// TIA Portal V19 export
FUNCTION "TetraPakV50_9" : Void   // FC118, STL
TITLE = Tetra Pak V50 IO-Link DeviceID 9 Process Data
{ S7_Optimized_Access := 'TRUE' }
AUTHOR : AFL
FAMILY : IO_Link
NAME : TP_V50_9
// Data words uses in function
// 
// HMI_CMD, dw X - command word from SCADA
// Bit 0 = auto
// Bit 1 = Manuel deactivate
// Bit 2 = Manuel activate
// Bit 3 = Locate
// Bit 4 = spare
// Bit 5 = spare
// Bit 6 = spare
// 
// HMI_INFO, dw X - info word to SCADA
// Bit 0  = activated
// Bit 1  = changing
// Bit 2  = faulty 
// Bit 3  = auto_man, Manuel = 1 
// Bit 4  = man_on_off
// Bit 5  = Reset_FB
// Bit 6  = ManualSelected
// Bit 7  = Set_FB
// Bit 8  = Locate Active 
// Bit 9  = spare 
// Bit 10 = spare 
// Bit 11 = spare  
// Bit 12 = spare 
// Bit 13 = spare 
// Bit 14 = fb_error - Alarm feedback error
// Bit 15 = spare 
// 
// Error status
// 0 (Everything is OK)
// 16 (Sensor target missing (#16))
// 17 (Setup prerequisite issue (#17))
// 18 (Pneumatic part issue (#18))
// 19 (Seat lift sensor issue (#19))
// 20 (Position not reached (#20))
// 21 (Unexpected movement (#21))
// 22 (Seat-lift sensor missing (#22))
// 23 (Pilot valve 1 missing (#23))
// 24 (Pilot valve 2 missing (#24))
// 25 (Pilot valve 3 missing (#25))
// 26 (Interlock active (#26))
// 27 (Output short circuit (#27))
// 28 (Setup aborted (#28))
// 29 (Blocked button (#29))
// 30 (Communication failure (#30))
// 31 (Safety stop active (#31))
// stored: AutoNumber false
   VAR_INPUT
      Addr : Int;   // First Byte address of 4 byte address space
      Pulse : Bool;   // Trigger one clean pulse on SV 1
      SV_1 : Bool;   // Trigger solenoid valve 1 for main valve activation
      Wink : Bool;   // Visual indication for locating the unit
   END_VAR
   VAR_OUTPUT
      ValvePosition : Real;   // Current Valve position (0 to 720 * 0.1)
      ValveState : Bool;   // Current Valve state
      O_DI4 : Bool;   // Output signal status Pin 4
      O_DI2 : Bool;   // Output signal status Pin 2
      Teach : Bool;   // Teach output for teach command bit
   END_VAR
   VAR_IN_OUT
      itemInfo : "ItemInfo_UDT";
      itemCommand : "ItemCommand_UDT";
      ErrorStatus : Byte;   // See Block Comment
      Main : Bool;   // Main energised Position
      DE_EN : Bool;   // De-Energized
      O_DA : Bool;   // Output device recognised
      O_DE : Bool;   // Output device error event has appeared
      O_PQ : Bool;   // Output port qualifer proces data valid
   END_VAR
   VAR_TEMP
      TW_Flag : Word;
      Tmp_ErrorStatus : Byte;   // Local Byte 6
      output : Bool;
   END_VAR
BEGIN

NETWORK
TITLE = Get items first byte address
// Get first byte address
      L     #Addr;
      SLW   3;
      LAR1;



NETWORK
TITLE = Valve Position
// Valve Position
      L     IW [AR1, P#0.0];
      DTR;
      L     0.1;
      *R;
      T     #ValvePosition;

// Error Status
      L     IB [AR1, P#2.0];
      T     #Tmp_ErrorStatus;
      SET;
      R     #Tmp_ErrorStatus.%X5;
      R     #Tmp_ErrorStatus.%X6;
      R     #Tmp_ErrorStatus.%X7;
      L     #Tmp_ErrorStatus;
      T     #ErrorStatus;


// ValveState
      L     IB [AR1, P#3.0];
      T     #TW_Flag;
      L     16;
      AW;
      L     16;
      ==I;
      =     #ValveState;


// Main
      L     IB [AR1, P#3.0];
      T     #TW_Flag;
      L     2;
      AW;
      L     2;
      ==I;
      =     #Main;

// DE_EN
      L     IB [AR1, P#3.0];
      T     #TW_Flag;
      L     1;
      AW;
      L     1;
      ==I;
      =     #DE_EN;

// PQI

      L     IB [AR1, P#4.0];
      T     #TW_Flag;

      L     #TW_Flag;
      L     1;
      AW;
      L     1;
      ==I;
      =     #O_DI4;



      L     #TW_Flag;
      L     2;
      AW;
      L     2;
      ==I;
      =     #O_DI2;

      L     #TW_Flag;
      L     32;
      AW;
      L     32;
      ==I;
      =     #O_DA;

      L     #TW_Flag;
      L     64;
      AW;
      L     64;
      ==I;
      =     #O_DE;


      L     #TW_Flag;
      L     128;
      AW;
      L     128;
      ==I;
      =     #O_PQ;

// *** Valve Fault Detected ***
      L     #ErrorStatus;
      L     1;
      >I;
      O;
      A     #O_DE;
      O;
      AN    #O_DA;
      AN    #O_DE;
      AN    #O_PQ;
      =     #itemInfo.fb_error;

// Pulse
      A     #Pulse;
      =     Q [AR1, P#0.2];  // Pulse output

// Valve Control

      AN    #itemInfo.auto_man;  // IF AUTO
//  A     "ACTIVATE"                  // AND ProcessReq
      A     #SV_1;
      O(;
      A     #itemInfo.auto_man;  // IF Manuel
      A     #itemInfo.man_on_off;  // Manuel on/off
      );
      =     Q [AR1, P#0.4];  // Set/reset Output
      =     #output;

// Locate

      A     #itemCommand.Locate;
      A     #itemInfo.LocateActive;
      R     Q [AR1, P#0.7];
      R     #itemCommand.Locate;


      A     #itemCommand.Locate;
      AN    #itemInfo.LocateActive;
      S     Q [AR1, P#0.7];
      R     #itemCommand.Locate;

// Teach

      A     #itemCommand.Teach;
      =     #Teach;

//****************** Outputs ************

      L     QB [AR1, P#0.0];
      T     QB [AR1, P#0.0];



NETWORK
TITLE = SCADA INFO & command
      AN    #itemCommand.Auto;
      AN    #itemCommand.Locate;
      AN    #itemCommand.Man_Act;
      AN    #itemCommand.Man_DeAct;
      AN    #itemCommand.Teach;
      AN    #itemCommand.SpareBool;
      AN    #itemCommand.SpareBool_1;
      AN    #itemCommand.SpareBool_2;
      AN    #itemCommand.SpareBool_3;
      AN    #itemCommand.SpareBool_4;
      AN    #itemCommand.SpareBool_5;
      AN    #itemCommand.SpareBool_6;
      AN    #itemCommand.SpareBool_7;
      AN    #itemCommand.SV_2SelectionBit;
      AN    #itemCommand.SV_3SelectionBit;
      AN    #itemCommand.SpareBool_10;
      JC    INFO;  // if commamd bits = 0 then no commands


      A     #itemCommand.Auto;
      R     #itemInfo.auto_man;
      JC    clea;

      A     #itemCommand.Man_DeAct;
      S     #itemInfo.auto_man;
      R     #itemInfo.man_on_off;
      JC    clea;

      A     #itemCommand.Man_Act;
      S     #itemInfo.auto_man;
      S     #itemInfo.man_on_off;
      JC    clea;
// Clear itemCommand word
clea: SET;
      R     #itemCommand.Auto;
      R     #itemCommand.Locate;
      R     #itemCommand.Man_Act;
      R     #itemCommand.Man_DeAct;
      R     #itemCommand.Teach;
      R     #itemCommand.SpareBool;
      R     #itemCommand.SpareBool_1;
      R     #itemCommand.SpareBool_2;
      R     #itemCommand.SpareBool_3;
      R     #itemCommand.SpareBool_4;
      R     #itemCommand.SpareBool_5;
      R     #itemCommand.SpareBool_6;
      R     #itemCommand.SpareBool_7;
      R     #itemCommand.SV_2SelectionBit;
      R     #itemCommand.SV_3SelectionBit;
      R     #itemCommand.SpareBool_10;
//clear command word

//;=========================== Scada info ================================
INFO: A     #itemInfo.fb_error;  // feedback error
      =     #itemInfo.faulty;
      A     #itemInfo.auto_man;
      =     #itemInfo.ManualSelected;  //Show Manual selected on SCADA
      A     #DE_EN;
      =     #itemInfo.Reset_FB;  //Show Reset FB in "Item Info & Operation" popup
      A     #Main;
      =     #itemInfo.Set_FB;  //Show Set FB in "Item Info & Operation" popup
      A     Q [AR1, P#0.7];
      =     #itemInfo.LocateActive;


//;                     // ================================
//;                     // = SET FB , SET/RES FB =
// Goto Changing
      A     #output;  // IF Output
      A     #Main;  // AND SetFB
      JC    ACT;  // Goto Activated
      A     #output;  // IF Output
      AN    #DE_EN;  // AND NOT SetFB
      JC    CHAN;
      JU    DEAC;
//;                     // ================================
//;                     // ================================
DEAC: R     #itemInfo.activated;  // Update = deactivated
      R     #itemInfo.changing;
      JU    NEX4;  //NEXT;
//;                     // ================================
CHAN: R     #itemInfo.activated;  // Update = activated
      S     #itemInfo.changing;
      JU    NEX4;  //NEXT;
//;                     // ================================
ACT:  S     #itemInfo.activated;  // Update = activated
      R     #itemInfo.changing;
      JU    NEX4;  //NEXT;
//;                     // ================================
NEX4: NOP   0;


END_FUNCTION
